# B&R Automation Studio project Cortadora_mappMotion
Automation Studio 4.12.2.93; technology packages: mapp 5.20.0, mappCockpit 5.20.0, mappMotion 5.20.2, mappView 5.20.0

## Configuration AcpTest

CPU 4PPC70.0702-20B, AutomationRuntime B4.91, Build 4.1.2, Safety 0.0, Vc V4.72.9

### Task classes (Cpu.sw)
```
Libraries: NcGlobal, sys_lib, brsystem, runtime
```

### Hardware
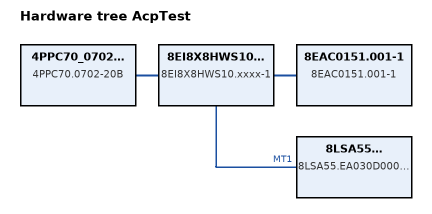
```
4PPC70_0702_20B : 4PPC70.0702-20B v1.5.4.0
  Connector IF2:
    ActivateDevice = 1
  ConfigurationID = Cortadora_mappMotion_AcpTest
  TimerDeviceType = EPLX2X
  TimerDevice = 4PPC70_0702_20B.IF1
  TaskClassIdleTime = 2000
  FileDevice1
  FileDeviceName1 = USER
  FileDevicePath1 = USER_PATH
  KeyMappingFile = VC\4PPC70_0702_20B.dis
8EAC0151.001-1 : 8EAC0151.001-1 v2.2.1.0  [SS -> 8EI8X8HWS10.xxxx-1.SS1]
8EI8X8HWS10.xxxx-1 : 8EI8X8HWS10.xxxx-1 v2.3.1.1  [PLK1 -> 4PPC70_0702_20B.IF1 (NodeNumber=1) [Cable Type=PowerlinkCable, Length=10, Version=1.0.0.3]]
  MotionTP = Acp10Arnc0
  BothEndSwitchesAreNormallyOpen_r1 = on
  QuickStopIsNormallyOpen_r1 = on
8LSA55.EA030D000-1 : 8LSA55.EA030D000-1 v1.0.6.40  [MT -> 8EI8X8HWS10.xxxx-1.MT1]
```

### Acp10cfg.ncc - 4PPC70_0702_20B/Motion/Acp10cfg.ncc
```
NcConfiguration (Version=5.20.1, NcSwId=Acp10)
  ACP10CF1_typ:
    cnt_nettrc_rec_drive = 1500
    bufsize_trace_upload = 1200
    tc_nc_man_task = Cyclic #1
    glob_pv_as_ncobject = Yes
    ncsys_dl_broadcast = Yes
    ncsys_dl_acp_reset = Yes
    safemc_log_err_to_ax = Yes
    network_init:
      ncsw_init_execute = Yes
      automatic_execute = No
      node_nr_warning = Yes
      net_err_before_ncact = Yes
    nettrc:
      enter_parsecrec = Yes
      enter_ncaction = Yes
      save_ring_startidx = Yes
    cam_prof_download:
      cam_dat_dl_parallel = No
      tc_cam_dl_parallel = Task class for NC Manager task
    plk_if[0]:
      if_name = IF1
      tc_CycDat_PLCopen = Task class for NC Manager task
      mc_broadcast_extdat = No
```

### Acp10map.ncm - 4PPC70_0702_20B/Motion/Acp10map.ncm
```
NcMapping (NcSwId=Acp10)
  NcObject gAxis01 (ModuleId=8EI8X8HWS10.xxxx-1, Type=ncAXIS, Channel=1, AcoposSimulation=Off, InitParameter=gAxis01i, AcoposParameter=gAxis01a, Disabled=FALSE, ModuleDisabled=FALSE)
  NcObject 8EI8X8HWS10.xxxx-1_ncV_AXIS1 (ModuleId=8EI8X8HWS10.xxxx-1, Type=ncV_AXIS, Channel=1, Disabled=TRUE, ModuleDisabled=FALSE)
```

## Configuration Config1

CPU 4PPC70.0573-20B, AutomationRuntime B4.91, Build 4.1.2, Safety 0.0, Vc V4.72.6

### Task classes (Cpu.sw)
```
Cyclic#1 (cycle 1600 us, tolerance 0 us):
  MotionCtrl <- MotionCtrl.prg
Cyclic#2 (cycle 11200 us, tolerance 22400 us):
  IMA_Client <- DataHandling.IMA_Client.prg
  VarExchang <- DataHandling.VarExchange.prg
Cyclic#3 (cycle 49600 us, tolerance 49600 us):
  ReadPar <- ReadPar.prg
Cyclic#8 (cycle 9600 us):
  VisuCtrl <- VisuCtrl.prg
DataObjects: DataMap <- DataHandling.DataMap.dob, McAcpSys
NcDataObjects: AcpParTab <- AcpParTab.dob, McDriveLog
VcDataObjects: Visu1 <- Visu.dob
Binaries: vccdt, McAcpSim, vccline, vcfile, arial, vctcal, vccbmp, arsvcreg, vccstr, vcbclass, vccbtn, vcmgr, vcgclass, vcdsint, vcnet, McProfGen, vcchtml, McAcpDrv, vcshared, arflatprv, vccddbox, vcxml, vccnum, vcpdvnc, FWRules, arcoal, vccalarm, vccurl, vcpfar00, vccbar, vcctext, vcpdsw, vcfntttf, vccovl, vccshape, vcalarm, vcpkat, vcctrend, udbdef, vccpopup, vcdsloc, vcrt, TCData, Visu102, Visu101, Visu103, vcpdi815, vcptelo, vcpdihd, vcpk, vcpfppc7, vcpdi855, arconfig, asfw, Cutter, Role, Config_2, ashwd, ExtEncod, iomap, MotionCfg, Config, ashwac, sysconf, User, robot2cm, Visu03, Visu01, Visu02, Visu
Libraries: MpBase, MpAlarmX, astime, runtime, standard, CoTrace, AsZip, FileIO, AsMath, McBase, MpAxis, McPureVAx, McAcpPar, McAcpAx, McAxis, McAxGroup, AsIMA, DataObj, inaclnt, sys_lib, brsystem, asieccon, powerlnk, vcresman, asepl
```

### Hardware
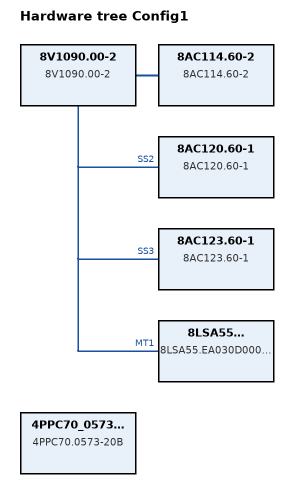
```
4PPC70_0573_20B : 4PPC70.0573-20B v1.5.4.0
  Connector IF1:
    CycleTime = 800
  Connector IF2:
    ActivateDevice = 1
    Mode = Manual
    InternetAddress = 192.168.0.25
    SubnetMask = 255.255.255.0
    Vnc1
    VncVcObjectName1 = Visu1
    VncKeyMappingFile1 = VC\PS2-Keyboard.dis
    ActivateSnmp = 2
  ConfigurationID = Cortadora_mappMotion_Config1
  UserPartitionSize = 0
  RemanentGlobalPvSize = 100
  EnableUsbRemoteInstall = 1
  TimerDeviceType = EPLX2X
  TimerDevice = 4PPC70_0573_20B.IF1
  TaskClassIdleTime = 800
  Cyclic1Duration = 1600
  Cyclic1Tolerance = 0
  Cyclic1Stack = 81920
  Cyclic2Duration = 11200
  Cyclic2Tolerance = 22400
  Cyclic3Duration = 49600
  Cyclic3Tolerance = 49600
  Cyclic8Duration = 9600
  FileDevice1
  FileDeviceName1 = USER
  FileDevicePath1 = USER_PATH
  TimeZone = 45
  ActivateOpcUa = 1
  OpcUaInformationModels_PV_Version = 1
  VcObjectName = Visu1
  KeyMappingFile = VC\4PPC70_0573_20B.dis
8AC114.60-2 : 8AC114.60-2 v1.0.0.8  [SS -> 8V1090.00-2.SS1; PLK1 -> 4PPC70_0573_20B.IF1 (NodeNumber=2) [Cable Type=PowerlinkCable, Length=10, Version=1.0.0.3]]
8AC120.60-1 : 8AC120.60-1 v2.2.0.0  [SS -> 8V1090.00-2.SS2]
  PlugInType = Encoder
  McAcoposTypeID = AcoposPlugInConfig
8AC123.60-1 : 8AC123.60-1 v2.2.0.0  [SS -> 8V1090.00-2.SS3]
  PlugInType = Encoder
  McAcoposTypeID = AcoposPlugInConfig
  LinesPerRevolution = 5000
  IgnoreCheck = 0
8LSA55.EA030D000-1 : 8LSA55.EA030D000-1 v1.0.4.40  [MT -> 8V1090.00-2.MT1]
8V1090.00-2 : 8V1090.00-2 v2.2.0.0
  DriveConfiguration/Module:
    McAcoposTypeID = AcoposConfig
    ActivateACOPOSSimulationOnPLC = 0
  DriveConfiguration/Channel[1]/RealAxis:
    AxisReference = Cutter
    MechanicalElementsIsInvisible = 0
  DriveConfiguration/Channel[1]/RealAxis/MechanicalElements/Gearbox:
    InputIsReadOnly = 0
    Input = 1
    OutputIsReadOnly = 0
    Output = 1
  DriveConfiguration/Channel[1]/RealAxis/MechanicalElements/RotaryToLinearTransformation:
    ReferenceDistanceIsReadOnly = 0
    ReferenceDistance = 1
  DriveConfiguration/Channel[1]/RealAxis/Controller:
    ModeIsReadOnly = 0
    Mode = PositionController
  DriveConfiguration/Channel[1]/RealAxis/Controller/Mode/Position:
    ProportionalGain = 43
    IntegrationTime = 0.0
    PredictionTime = 0.0004
    TotalDelayTime = 0.0004
  DriveConfiguration/Channel[1]/RealAxis/Controller/Mode/Speed:
    ProportionalGainIsReadOnly = 0
    ProportionalGain = 0.4
    IntegrationTimeIsReadOnly = 0
    IntegrationTime = 0.0
    FilterTimeIsReadOnly = 0
    FilterTime = 0.0
  DriveConfiguration/Channel[1]/RealAxis/Controller/Mode/LoopFilters:
    LoopFilterXIsReadOnly = 0
    LoopFilter1 = NotUsed
    LoopFilter2 = NotUsed
    LoopFilter3 = NotUsed
  DriveConfiguration/Channel[1]/RealAxis/Homing:
    ModeIsReadOnly = 0
    Mode = Absolute
  DriveConfiguration/Channel[1]/RealAxis/Homing/Mode:
    Position = -300
  DriveConfiguration/Channel[1]/RealAxis/Homing:
    RestorePositionVariable = 
  DriveConfiguration/Channel[1]/RealAxis/StopReaction:
    QuickstopIsReadOnly = 0
    Quickstop = DecelerationLimit
    DriveErrorIsReadOnly = 0
    DriveError = DecelerationLimit
  DriveConfiguration/Channel[1]/RealAxis/MovementErrorLimits:
    PositionError = 100000000
    VelocityErrorMonitoring = NotUsed
  DriveConfiguration/Channel[1]/RealAxis:
    JerkFilterIsReadOnly = 0
    JerkFilter = NotUsed
  DriveConfiguration/Channel[1]/RealAxis/DigitalInputs/HomingSwitch:
    SourceIsReadOnly = 0
    Source = Force
    Level = High
  DriveConfiguration/Channel[1]/RealAxis/DigitalInputs/PositiveLimitSwitch:
    Source = Force
    Level = High
  DriveConfiguration/Channel[1]/RealAxis/DigitalInputs/NegativeLimitSwitch:
    Source = Force
    Level = High
  DriveConfiguration/Channel[1]/RealAxis/DigitalInputs/Trigger1:
    Source = X1Trigger1
    Level = High
  DriveConfiguration/Channel[1]/RealAxis/DigitalInputs/Trigger2:
    Source = X1Trigger2
    Level = High
  DriveConfiguration/Channel[1]/RealAxis/DigitalInputs/Quickstop:
    Input = NotUsed
  DriveConfiguration/Channel[1]/RealAxis/Simulation:
    SimulationModeOnPLC = SetValueGeneration
    SimulationModeOnACOPOS = NotUsed
  DriveConfiguration/Channel[1]:
    ExternalEncoderAxis = Used
  DriveConfiguration/Channel[1]/ExternalEncoderAxis:
    AxisReference = ExtEncod
  DriveConfiguration/Channel[1]/ExternalEncoderAxis/EncoderLink:
    PositionEncoder = EncoderSS3X11
    PositionFilter = ExtrapolationAndDisturbance
  DriveConfiguration/Channel[1]/ExternalEncoderAxis/EncoderLink/PositionFilter:
    PositionFilterTimeConstant = 0.2
    ExtrapolationTime = 0.1
  DriveConfiguration/Channel[1]/ExternalEncoderAxis:
    MechanicalElementsIsInvisible = 0
  DriveConfiguration/Channel[1]/ExternalEncoderAxis/MechanicalElements/Gearbox:
    InputIsReadOnly = 0
    Input = 1
    OutputIsReadOnly = 0
    Output = 1
  DriveConfiguration/Channel[1]/ExternalEncoderAxis/MechanicalElements/RotaryToLinearTransformation:
    ReferenceDistanceIsReadOnly = 0
    ReferenceDistance = 314.159
  DriveConfiguration/Channel[1]/ExternalEncoderAxis/Homing:
    Mode = Direct
  DriveConfiguration/Channel[1]/ExternalEncoderAxis/Homing/Mode:
    Position = 0.0
    ReferencePulse = NotUsed
  DriveConfiguration/Channel[1]/ExternalEncoderAxis/Homing:
    RestorePositionVariable = 
  DriveConfiguration/Channel[1]/ChannelFeatures:
    FeatureRef[1] = Feature_AcpParTable
```

### Cutter.axis - 4PPC70_0573_20B/mappMotion/Cutter.axis
```
Element Cutter (Type=axis)
  BaseTypeIsReadOnly = 0
  BaseType = RotaryPeriodic
    MeasurementUnitIsReadOnly = 0
    MeasurementUnit = 17476
    MeasurementResolutionIsReadOnly = 0
    MeasurementResolution = 0.01
    CountDirectionIsReadOnly = 0
    CountDirection = Inverse
    PeriodSettings:
      Period = 360.0
  MovementLimitsIsReadOnly = 0
  MovementLimits = Internal
    Position:
      LowerLimitMin = -1.79769313486231E308
      UpperLimitMax = 1.79769313486231E308
      LowerLimit = -1000.0
      UpperLimit = 1000.0
    VelocityIsReadOnly = 0
    Velocity:
      VelocityMax = 3.4E38
      Velocity = 3000000
    AccelerationIsReadOnly = 0
    Acceleration:
      AccelerationMax = 3.4E38
      Acceleration = 5000000000000
    DecelerationIsReadOnly = 0
    Deceleration:
      DecelerationMax = 3.4E38
      Deceleration = 5000000000000
  Alarms = MpAlarmX
```

## Configuration P3wC70

CPU 4PPC70.0702-20B, AutomationRuntime B4.91, Build 4.1.2, Safety 0.0, Vc V4.72.6

### Task classes (Cpu.sw)
```
Cyclic#1 (cycle 1600 us, tolerance 0 us):
  MotionCtrl <- MotionCtrl.prg
  IMA_Client <- DataHandling.IMA_Client.prg
  VarExchang <- DataHandling.VarExchange.prg
Cyclic#3 (cycle 49600 us, tolerance 49600 us):
  ReadPar <- ReadPar.prg
Cyclic#8 (cycle 9600 us):
  VisuCtrl <- VisuCtrl.prg
DataObjects: DataMap <- DataHandling.DataMap.dob, McAcpSys
NcDataObjects: AcpParTab <- AcpParTab.dob, McDriveLog
VcDataObjects: Visu_7 <- Visu_7inch.dob
Binaries: vccdt, vccline, vcfile, vcptelo, vctcal, Visu_702, vccddbox, vccbmp, arsvcreg, vccstr, vcbclass, vccbtn, vcmgr, vcgclass, vcdsint, vcnet, McProfGen, vcchtml, vcpdihd, vcshared, arflatprv, vcxml, vccnum, vcpdvnc, FWRules, vccovl, vcpdi855, arcoal, vccalarm, vccurl, vccbar, vcpfppc7, vcctext, Visu_703, vcpdsw, vcfntttf, McAcpDrv, vccshape, vcalarm, vccpopup, vcpkat, vcctrend, udbdef, vcpdi815, vcdsloc, Visu_701, vcpk, vcrt, TCData, McAcpSim, arial, arconfig, Alarms, asfw, Cutter, Role, ashwd, iomap, MotionCfg, ashwac, sysconf, User, Config_1, ExtEncod, Config_2, Config, robotevi, robot2cm, vcpfar00, Config_4, Virtual
Libraries: MpBase, MpAlarmX, astime, runtime, CoTrace, AsZip, FileIO, asieccon, powerlnk, vcresman, sys_lib, dataobj, asepl, standard, mcbase, mcaxis, mcacpax, mpaxis
```

### Hardware
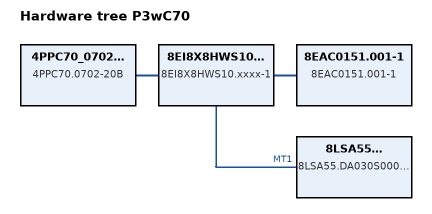
```
4PPC70_0702_20B : 4PPC70.0702-20B v1.5.4.0
  Connector IF1:
    CycleTime = 800
    Mode = CN
    NodeID = 3
    InaNodeNumber = 3
  Connector IF2:
    ActivateDevice = 1
    Mode = Manual
    InternetAddress = 192.168.0.25
    SubnetMask = 255.255.255.0
    Vnc1
    VncVcObjectName1 = Visu_7
    VncKeyMappingFile1 = VC\PS2-Keyboard.dis
    ActivateSnmp = 2
  ConfigurationID = Cortadora_mappMotion_P3
  ConfigVersion = 5.0.0
  UserPartitionSize = 0
  RemanentGlobalPvSize = 1000
  EnableUsbRemoteInstall = 1
  TimerDeviceType = EPLX2X
  TimerDevice = 4PPC70_0702_20B.IF1
  TaskClassIdleTime = 1600
  Cyclic1Duration = 1600
  Cyclic1Tolerance = 0
  Cyclic1Stack = 81920
  Cyclic3Duration = 49600
  Cyclic3Tolerance = 49600
  Cyclic8Duration = 9600
  FileDevice1
  FileDeviceName1 = USER
  FileDevicePath1 = USER_PATH
  VcObjectName = Visu_7
  KeyMappingFile = VC\4PPC70_0702_20B.dis
8EAC0151.001-1 : 8EAC0151.001-1 v2.2.1.0  [SS -> 8EI8X8HWS10.xxxx-1.SS1]
  PlugInType = Encoder
  McAcoposTypeID = AcoposP3PlugInSConfig
  InterfaceType = IncrementalEAC151
  LineResistance = SpecifyValue
  Value = 0.0
  Symmetry = Symmetrical
  LineTermination = 0
  ReferencePulseDetection = 0
  LineCount = 5000
  MaxExpectedOutputFrequency = 200
8EI8X8HWS10.xxxx-1 : 8EI8X8HWS10.xxxx-1 v2.3.1.1  [PLK1 -> 4PPC70_0702_20B.IF1 (NodeNumber=2) [Cable Type=PowerlinkCable, Length=10, Version=1.0.0.3]]
  EnableDNA = on
  DriveConfiguration/Module:
    McAcoposTypeID = AcoposP3DConfig
    ActivateACOPOSSimulationOnPLC = 0
  DriveConfiguration/Encoder/EncoderX41:
    InterfaceType = EnDat
  DriveConfiguration/Channel[1]/RealAxis:
    AxisReference = Cutter
    MechanicalElementsIsInvisible = 0
  DriveConfiguration/Channel[1]/RealAxis/MechanicalElements/Gearbox:
    InputIsReadOnly = 0
    Input = 1
    OutputIsReadOnly = 0
    Output = 1
  DriveConfiguration/Channel[1]/RealAxis/MechanicalElements/RotaryToLinearTransformation:
    ReferenceDistanceIsReadOnly = 0
    ReferenceDistance = 1
  DriveConfiguration/Channel[1]/RealAxis/Controller:
    ModeIsReadOnly = 0
    Mode = PositionControllerWithTorqueFeedForward
  DriveConfiguration/Channel[1]/RealAxis/Controller/Mode/Position:
    ProportionalGainIsReadOnly = 0
    ProportionalGain = 60
    IntegrationTimeIsReadOnly = 0
    IntegrationTime = 0.0
    TotalDelayTime = 0.0004
  DriveConfiguration/Channel[1]/RealAxis/Controller/Mode/Speed:
    ProportionalGainIsReadOnly = 0
    ProportionalGain = 0.9
    IntegrationTimeIsReadOnly = 0
    IntegrationTime = 0.0
    FilterTimeIsReadOnly = 0
    FilterTime = 0.0
  DriveConfiguration/Channel[1]/RealAxis/Controller/Mode:
    FeedForwardIsReadOnly = 0
    FeedForward = Standard
  DriveConfiguration/Channel[1]/RealAxis/Controller/Mode/FeedForward:
    TorqueLoad = 0.0
    TorquePositive = 0.008
    TorqueNegative = 0.00355563
    SpeedTorqueFactor = 0.0109247
    Inertia = 0.00221627
    AccelerationFilterTime = 0.0
  DriveConfiguration/Channel[1]/RealAxis/Controller/Mode/LoopFilters:
    LoopFilterXIsReadOnly = 0
    LoopFilter1 = NotUsed
    LoopFilter2 = NotUsed
    LoopFilter3 = NotUsed
  DriveConfiguration/Channel[1]/RealAxis/Homing:
    ModeIsReadOnly = 0
    Mode = Absolute
  DriveConfiguration/Channel[1]/RealAxis/Homing/Mode:
    Position = -300
  DriveConfiguration/Channel[1]/RealAxis/Homing:
    RestorePositionVariable = 
  DriveConfiguration/Channel[1]/RealAxis/StopReaction:
    QuickstopIsReadOnly = 0
    Quickstop = DecelerationLimit
    DriveErrorIsReadOnly = 0
    DriveError = DecelerationLimit
  DriveConfiguration/Channel[1]/RealAxis/MovementErrorLimits:
    PositionError = 10000
    VelocityErrorMonitoring = NotUsed
  DriveConfiguration/Channel[1]/RealAxis:
    JerkFilterIsReadOnly = 0
    JerkFilter = NotUsed
  DriveConfiguration/Channel[1]/RealAxis/DigitalInputs/HomingSwitch:
    SourceIsReadOnly = 0
    Source = Force
    Level = High
  DriveConfiguration/Channel[1]/RealAxis/DigitalInputs/PositiveLimitSwitch:
    SourceIsReadOnly = 0
    Source = Force
    Level = High
  DriveConfiguration/Channel[1]/RealAxis/DigitalInputs/NegativeLimitSwitch:
    SourceIsReadOnly = 0
    Source = Force
    Level = High
  DriveConfiguration/Channel[1]/RealAxis/DigitalInputs/Trigger1:
    Source = X8Trigger1
    Level = High
  DriveConfiguration/Channel[1]/RealAxis/DigitalInputs/Trigger2:
    Source = X8Trigger2
    Level = High
  DriveConfiguration/Channel[1]/RealAxis/DigitalInputs/Quickstop:
    Input = NotUsed
  DriveConfiguration/Channel[1]/RealAxis/Simulation:
    SimulationModeOnPLC = SetValueGeneration
    SimulationModeOnACOPOS = NotUsed
  DriveConfiguration/Channel[1]:
    ExternalEncoderAxis = Used
  DriveConfiguration/Channel[1]/ExternalEncoderAxis:
    AxisReference = ExtEncod
  DriveConfiguration/Channel[1]/ExternalEncoderAxis/EncoderLink:
    PositionEncoder = EncoderX41x
    PositionFilter = ExtrapolationAndDisturbance
  DriveConfiguration/Channel[1]/ExternalEncoderAxis/EncoderLink/PositionFilter:
    PositionFilterTimeConstant = 0.0
    ExtrapolationTime = 0.1
  DriveConfiguration/Channel[1]/ExternalEncoderAxis:
    MechanicalElementsIsInvisible = 0
  DriveConfiguration/Channel[1]/ExternalEncoderAxis/MechanicalElements/Gearbox:
    InputIsReadOnly = 0
    Input = 1
    OutputIsReadOnly = 0
    Output = 1
  DriveConfiguration/Channel[1]/ExternalEncoderAxis/MechanicalElements/RotaryToLinearTransformation:
    ReferenceDistanceIsReadOnly = 0
    ReferenceDistance = 31.4159
  DriveConfiguration/Channel[1]/ExternalEncoderAxis/Homing:
    Mode = Direct
  DriveConfiguration/Channel[1]/ExternalEncoderAxis/Homing/Mode:
    Position = 0.0
    ReferencePulse = NotUsed
  DriveConfiguration/Channel[1]/ExternalEncoderAxis/Homing:
    RestorePositionVariable = 
8LSA55.DA030S000-3 : 8LSA55.DA030S000-3 v2.2.0.1  [MT -> 8EI8X8HWS10.xxxx-1.MT1]
  M1/MotorParameters:
    MOTOR_AMB_TEMP_RATED = 40
```

### ExtEncod.axis - 4PPC70_0702_20B/mappMotion/ExtEncod.axis
```
Element ExtEncod (Type=axis)
  BaseTypeIsReadOnly = 0
  BaseType = Linear
    MeasurementUnit = 5066068
    MeasurementResolutionIsReadOnly = 0
    MeasurementResolution = 0.01
    CountDirectionIsReadOnly = 0
    CountDirection = Inverse
  MovementLimitsIsReadOnly = 0
  MovementLimits = Internal
    Position:
      LowerLimitMin = -1.79769313486231E308
      UpperLimitMax = 1.79769313486231E308
      LowerLimit = -1000.0
      UpperLimit = 1000.0
    VelocityIsReadOnly = 0
    Velocity:
      VelocityMax = 3.4E38
      Velocity = 1000
    AccelerationIsReadOnly = 0
    Acceleration:
      AccelerationMax = 3.4E38
      Acceleration = 10000
    DecelerationIsReadOnly = 0
    Deceleration:
      DecelerationMax = 3.4E38
      Deceleration = 10000
  Alarms = MpAlarmX
```

### MotionCfg.mappmotioncfg - 4PPC70_0702_20B/mappMotion/MotionCfg.mappmotioncfg
```
Element MappMotionConfiguration (Type=mappmotioncfg)
  Processing:
    ProcessingTaskClass = 1
  SharedAlarms:
    Axis = MpAlarmX
```

## Logical view

Binary libraries used (declarations not repeated): operator, runtime, astime, AsIecCon, standard, AsZip, FileIO, AsMath, NcGlobal 5.20.1, sys_lib, brsystem, MpBase, MpAlarmX 5.20.0, CoTrace, McBase, MpAxis, McPureVAx 5.20.2, McAcpPar 5.20.2, McAcpAx, McAxis, McAxGroup 5.20.2, AsIMA, DataObj, inaclnt

### Global.typ - Global data types
```iecst
TYPE
	gCutter_enum :
		(
		Default,
		Encoder,
		Time,
		Sensor,
		Speed,
		EncoderDieCutter,
		SensorDieCutter
		);
	DataCollector_state_enum :
		(
		ST_IDLE,
		ST_CONNECTING,
		ST_CONNECTED,
		ST_CLOSE_CONNECTION,
		ST_ERROR_ACTIVE,
		ST_RESET_ERROR
		);
END_TYPE
```

### Global.var - Global variables
```iecst
VAR
	MODE_SELECTED : gCutter_enum;
	posTroqueladora : LREAL;
	SensorSignal : BOOL;
	MachineStateIndex : UINT := 0;
	MachineInOperation : BOOL;
	MachineInitializing : BOOL;
	MachineAutotuning : BOOL;
	MachineHoming : BOOL;
	MachineReady : BOOL;
	CurrentPage : INT;
END_VAR
VAR RETAIN
	HMI_MODE_SELECTED : gCutter_enum;
END_VAR
VAR
	TotalCutsPerMode : LREAL;
	BoxIsOpen : BOOL;
	CycleTime : REAL := 1.6;
	MinuteInMiliseconds : DINT := 60000;
	CycleTimeSum : REAL;
	CutsPerMinute_Distance : REAL;
	CutsPerMinute_Time : REAL;
	CutsPerMinute_Sensor : REAL;
	cutEnabled : BOOL; (*Info proveniente de la troqueladora*)
	auxToCut : BOOL;
	encActPosPerRev : DINT;
	actPosExtEncoder : LREAL; (*Info proveniente de la troqueladora*)
	oneCutEncoderCutterDieCmd : BOOL;
END_VAR
```


### Program Logical/MotionCtrl (IEC)

#### Main.st - Init, cyclic, exit code
```iecst
PROGRAM _INIT
	(* Insert code here *)
	MpAxisBasic_Cutter.MpLink := ADR(Cutter);
	MpAxisBasic_Cutter.Parameters := ADR(MpAxisBasicPar_Cutter);

	MpAxisBasicPar_Cutter.Velocity := DefaultVelocity;
	MpAxisBasicPar_Cutter.Acceleration := DefaultAcceleration;
	MpAxisBasicPar_Cutter.Deceleration := DefaultDeceleration;
	MpAxisBasicPar_Cutter.Distance := DefaultDistance;
	MpAxisBasicPar_Cutter.Position := DefaultPosition;

	MC_BR_InitHome_AcpAx_0.Axis := ADR(Cutter);
	MC_BR_InitHome_AcpAx_0.HomingParameters := McAcpAxHomingPar_0;
	McAcpAxHomingPar_0.HomingMode := InitHomingMode;

	MC_BR_InitHome_AcpAx_0.Axis := ADR(Cutter);
	MC_BR_InitHome_AcpAx_0.HomingParameters.HomingMode := InitHomingMode;
	MC_BR_InitHome_AcpAx_0.HomingParameters.Position := DefaultPosition;
	MC_BR_InitHome_AcpAx_0.HomingParameters.StartVelocity := 50;
	MC_BR_InitHome_AcpAx_0.HomingParameters.HomingVelocity := 50;
	MC_BR_InitHome_AcpAx_0.HomingParameters.Acceleration := 500;
	MC_BR_InitHome_AcpAx_0.HomingParameters.SwitchEdge := 0;
	MC_BR_InitHome_AcpAx_0.HomingParameters.StartDirection := 1;
	MC_BR_InitHome_AcpAx_0.HomingParameters.HomingDirection := 0;

	MpAxisBasicPar_Cutter.Homing.Mode := HomingMode;
	MpAxisBasicPar_Cutter.Homing.Position := DefaultPosition;

	//Autotune settings
	MpAxisBasicPar_Cutter.AutoTune.MaxCurrentPercent := 75;
	MpAxisBasicPar_Cutter.AutoTune.MaxDistance := 5;
	MpAxisBasicPar_Cutter.AutoTune.MaxPositionError := 2000;

	(*//Reading external encoder
	MC_BR_CyclicProcessParID_AcpAx_0.Axis := ADR(ExtEncod);
	MC_BR_CyclicProcessParID_AcpAx_0.DataAddress := ADR(McAcpAxCycParID_0);
	MC_BR_CyclicProcessParID_AcpAx_0.Mode := mcACPAX_CYCLIC_PARID_READ;
	MC_BR_CyclicProcessParID_AcpAx_0.NumberOfParIDs := 1;

	McAcpAxCycParID_0.DataType:= mcACPAX_PARTYPE_DINT;
	McAcpAxCycParID_0.ParID := 246;//423 Actual Position, 246 Actual Position per Revolution
	McAcpAxCycParID_0.RefreshMode := mcACPAX_CYCLIC_EVERY_RECORD;
	McAcpAxCycParID_0.VariableAddress := ADR(EncoderActPos);*)

	MpAxisBasic_Cutter.Enable := TRUE;

END_PROGRAM

PROGRAM _CYCLIC

	Pulses := REAL_TO_UINT(HMIPulses * 4);

	vAxisEncoderActPos;
	//Basic calculation of encoder perimeter adjusted via HMI
	EncoderPerimeter := (amPI * EncoderDiameter);

	//Cutting Offset - Not used
	DelayTimer_0.PT := UDINT_TO_TIME(SensorCutDelay);

	//mapping for visu
	BoxIsOpen := NOT MpAxisBasic_Cutter.Info.DigitalInputsStatus.DriveEnable;

	CASE MODE_SELECTED OF

		Default:

			InitAxis;

			CutterTimer.IN := FALSE;
			CutterTimer.PT := DINT_TO_TIME(0);

		Encoder:

			MpAxisBasicPar_Cutter.Velocity := DefaultVelocity;
			MpAxisBasicPar_Cutter.Acceleration := DefaultAcceleration;
			MpAxisBasicPar_Cutter.Deceleration := DefaultDeceleration;

			//Start Encoder Position Reading
			//MC_BR_CyclicProcessParID_AcpAx_0.Enable := TRUE;
			//EncoderActPos := encActPosPerRev;
			encActPosPerRev;

			IF CorrectDistance THEN
				ActualProductLength := HMICuttingLength + (CuttingOffset *-1);
				CorrectionFactor := (HMICuttingLength/ActualProductLength);
				HMICorrectionFactorPercentage := (CorrectionFactor *100) - 100;
				CuttingOffset := 0;
				CorrectDistance := FALSE;
			END_IF;

			HMICorrectionFactorMilimeters :=((HMICorrectionFactorPercentage/100) * HMICuttingLength);

			IF ClockwiseCount THEN

				IF EDGEPOS(EncoderActPosOld > EncoderActPos) AND ((EncoderActPosOld - EncoderActPos) > (Pulses*0.995)) THEN
					FullTurnCount := FullTurnCount + 1;
				END_IF;

				PartOfTurn := (DINT_TO_REAL(EncoderActPos)/Pulses);

			ELSE

				IF EDGEPOS(EncoderActPos > EncoderActPosOld) AND ((EncoderActPos - EncoderActPosOld) > (Pulses*0.995)) THEN
					FullTurnCount := FullTurnCount + 1;
				END_IF;

				PartOfTurn := 1 - (DINT_TO_REAL(EncoderActPos)/Pulses);

			END_IF;

			IF PartOfTurn >= (0.99) OR PartOfTurn < 0 THEN
				PartOfTurn := 0;
			END_IF;

			RealTurns := FullTurnCount + PartOfTurn;

			IF Empezar AND cutEnabled THEN

				MachineInOperation := TRUE;

				CycleTimeSum := CycleTimeSum + CycleTime;

				CountTurns;

				IF MpAxisBasic_Cutter.MoveDone THEN
					MpAxisBasic_Cutter.MoveAdditive := FALSE;
				END_IF;

				IF EDGEPOS(MpAxisBasic_Cutter.MoveDone) THEN
					NumberOfCuts_Distance := NumberOfCuts_Distance + 1;
				END_IF;

				RemainingDistance := ((NeededTurns - RealTurns) * EncoderPerimeter);
				TraveledDistance := HMICuttingLength - RemainingDistance;

				HMITraveledDistance := TraveledDistance ;
				HMIRemainingDistance := RemainingDistance;

				MC_BR_CyclicProcessParID_AcpAx_0();

				IF MpAxisBasic_Cutter.Error THEN
					MpAxisBasic_Cutter.MoveAdditive := FALSE;
					MpAxisBasic_Cutter.ErrorReset := TRUE;
				ELSE
					MpAxisBasic_Cutter.ErrorReset := FALSE;
				END_IF;

			END_IF;

			IF NOT Empezar THEN

				HMITraveledDistance := 0 ;
				HMIRemainingDistance := 0;
				CurrentProductTurns := 0;
				NeededTurns := 0;

				MC_BR_CyclicProcessParID_AcpAx_0.Enable := FALSE;

			END_IF;

			TotalCutsPerMode := NumberOfCuts_Distance;

		Time:

			MpAxisBasicPar_Cutter.Velocity := DefaultVelocity;
			MpAxisBasicPar_Cutter.Acceleration := DefaultAcceleration;
			MpAxisBasicPar_Cutter.Deceleration := DefaultDeceleration;

			CycleTimeSum := CycleTimeSum + CycleTime;

			IF Empezar THEN

				MachineInOperation := TRUE;
				CycleTimeSum := CycleTimeSum + CycleTime;
				UserTime := REAL_TO_DINT(HMITime*1000);
				TimeIsOver := CutterTimer.Q;
				CutterTimer.PT := DINT_TO_TIME(UserTime);
				ElapsedTime := (TIME_TO_REAL(CutterTimer.ET)/1000);
				RemainingTime := (REAL_TO_DINT(HMITime) - ElapsedTime);

				IF TimeIsOver THEN
					DelayTimer_0.IN := TRUE;
					CutterTimer.IN := FALSE;
				ELSE
					CutterTimer.IN := TRUE;
				END_IF;

				IF MpAxisBasic_Cutter.MoveDone THEN
					MpAxisBasic_Cutter.MoveAdditive := FALSE;
				END_IF;

				IF EDGEPOS(MpAxisBasic_Cutter.MoveDone) THEN
					NumberOfCuts_Time := NumberOfCuts_Time + 1;
				END_IF;

			ELSE

				ElapsedTime := 0;
				RemainingTime := 0;

			END_IF;

			TotalCutsPerMode := NumberOfCuts_Time;
			CutsPerMinute_Time := (60/HMITime);

			CutterTimer();

		Sensor:

			MpAxisBasicPar_Cutter.Velocity := DefaultVelocity;
			MpAxisBasicPar_Cutter.Acceleration := DefaultAcceleration;
			MpAxisBasicPar_Cutter.Deceleration := DefaultDeceleration;

			CycleTimeSum := CycleTimeSum + CycleTime;

			IF Empezar AND cutEnabled THEN

				MachineInOperation := TRUE;
				SensorSignal := MpAxisBasic_Cutter.Info.DigitalInputsStatus.Trigger1;
				FilterTimer_0.PT := UINT_TO_TIME(FilterTime);

				IF NOT FilterActive THEN

					IF EDGEPOS(MpAxisBasic_Cutter.Info.DigitalInputsStatus.Trigger1 OR inputTest) OR auxToCut THEN
						auxToCut := FALSE;
						FilterTimer_0.IN := TRUE;
						DelayTimer_0.IN := TRUE;
						FilterActive := TRUE;
					END_IF;

				END_IF;

				IF FilterTimer_0.Q THEN
					FilterActive := FALSE;
					FilterTimer_0.IN := FALSE;
				END_IF;

				FilterActive := FilterTimer_0.IN;

				FilterTimer_0();

				IF MpAxisBasic_Cutter.MoveDone THEN
					MpAxisBasic_Cutter.MoveAdditive := FALSE;
					SensorSignal := FALSE;
				END_IF;

				IF EDGEPOS(MpAxisBasic_Cutter.MoveDone) THEN
					NumberOfCuts_Sensor := NumberOfCuts_Sensor + 1;
				END_IF;

			END_IF;

			TotalCutsPerMode := NumberOfCuts_Sensor;
			CutsPerMinute_Sensor := NumberOfCuts_Sensor/CycleTimeSum;
		Speed:

			MachineInOperation := TRUE;

			CycleTimeSum := CycleTimeSum + CycleTime;

			IF Empezar THEN

				MpAxisBasicPar_Cutter.Velocity := HMIRevolutionsPerSecond * UnitsPerRevolution;
				MpAxisBasicPar_Cutter.Acceleration := MpAxisBasicPar_Cutter.Velocity * 10;
				MpAxisBasicPar_Cutter.Deceleration := MpAxisBasicPar_Cutter.Velocity * 10;
				MpAxisBasic_Cutter.MoveVelocity := TRUE;

			ELSE

				IF NOT MpAxisBasic_Cutter.IsHomed THEN
					ManualMoveAbsolute := TRUE;
				END_IF;

				MpAxisBasic_Cutter.MoveVelocity := FALSE;

			END_IF;

			IF (MpAxisBasic_Cutter.Velocity <> MpAxisBasicPar_Cutter.Velocity) AND Empezar THEN
				MpAxisBasic_Cutter.Update := TRUE;
			END_IF;

			IF MpAxisBasic_Cutter.UpdateDone THEN
				MpAxisBasic_Cutter.Update := FALSE;
			END_IF;

	END_CASE;

	//Whenever the operator presses Manual Cut the motor should do a full turn unless there is an active movement
	IF ManualCut AND (MpAxisBasic_Cutter.Info.PLCopenState = AxisStandstill) THEN

		MpAxisBasic_Cutter.MoveAdditive := TRUE;

		IF MpAxisBasic_Cutter.MoveDone THEN
			MpAxisBasic_Cutter.MoveAdditive := FALSE;
			ManualCut := FALSE;
		END_IF;

	END_IF;

	//For Visu
	IF Empezar THEN

		Count := Count + 0.0016;
		IF CountOld > Count THEN
			MaxCount := CountOld;
		END_IF;

		CountOld := Count;

	ELSE

		MachineInOperation := FALSE;
		MpAxisBasic_Cutter.MoveVelocity := FALSE;
		MpAxisBasic_Cutter.MoveAdditive := FALSE;
		CycleTimeSum := 0;
		MaxCount := 0;
		Count := 0;

	END_IF;

	//Sum of total cuts
	IF EDGEPOS(MpAxisBasic_Cutter.MoveDone) THEN

		Count := 0;
		TotalCuts := TotalCuts + 1;

	END_IF;

	IF MaxCount = 0 THEN
		ProductionSpeed := 0;
	ELSE
		ProductionSpeed := 60/MaxCount;
	END_IF;

	TotalCurrentCuts := NumberOfCuts_Time + NumberOfCuts_Sensor + NumberOfCuts_Distance;

	IF ResetCutsPerMode THEN
		NumberOfCuts_Time := 0;
		NumberOfCuts_Sensor := 0;
		NumberOfCuts_Distance := 0;
		ResetCutsPerMode := FALSE;
	END_IF;

	IF ResetTotalCuts THEN

		TotalCuts := 0;
		ResetTotalCuts := FALSE;

	END_IF;

	//Manual Controls
	IF NOT Empezar AND NOT MpAxisBasic_Cutter.MoveActive AND (CurrentPage = 1) THEN

		IF ManualMoveAdditivePos THEN
			ManualMoveAdditivePos := FALSE;
			MpAxisBasic_Cutter.MoveAdditive := TRUE;
			MpAxisBasicPar_Cutter.Distance := HMIDistance;
		END_IF;

		IF ManualMoveAdditiveNeg THEN
			ManualMoveAdditiveNeg := FALSE;
			MpAxisBasic_Cutter.MoveAdditive := TRUE;
			MpAxisBasicPar_Cutter.Distance := HMIDistance * -1;
		END_IF;

		IF ManualMoveAbsolute THEN
			MpAxisBasic_Cutter.MoveAbsolute := TRUE;
			MpAxisBasicPar_Cutter.Position := HomePosition;
			MpAxisBasicPar_Cutter.Direction := 0;
		END_IF;

	END_IF;

	IF MpAxisBasic_Cutter.MoveDone THEN

		ManualMoveAdditivePos := FALSE;
		ManualMoveAdditiveNeg := FALSE;
		ManualMoveAbsolute := FALSE;
		MpAxisBasic_Cutter.MoveAdditive := FALSE;
		MpAxisBasic_Cutter.MoveAbsolute := FALSE;

	END_IF;

	IF DelayTimer_0.Q THEN

		DelayTimer_0.IN := FALSE;
		//MpAxisBasic_Cutter.MoveAdditive := TRUE;

	END_IF;

	IF (CurrentPage = 0) THEN

		MpAxisBasicPar_Cutter.Distance := DefaultDistance;
		MpAxisBasicPar_Cutter.Position := DefaultPosition;

	END_IF;

	IF NOT MpAxisBasic_Cutter.Info.DigitalInputsStatus.DriveEnable THEN

		Empezar := FALSE;
		MpAxisBasic_Cutter.Power := FALSE;
		MpAxisBasic_Cutter.Home := FALSE;
		MpAxisBasic_Cutter.MoveAdditive := FALSE;
		MpAxisBasic_Cutter.MoveAbsolute := FALSE;
		MpAxisBasic_Cutter.MoveVelocity := FALSE;
		ManualMoveAdditivePos := FALSE;
		ManualMoveAdditiveNeg := FALSE;
		ManualMoveAbsolute := FALSE;
		MODE_SELECTED := Default;

	ELSE

		MpAxisBasic_Cutter.Stop := FALSE;

	END_IF;

	IF MpAxisBasic_Cutter.Error THEN
		MpAxisBasic_Cutter.ErrorReset := TRUE;
	ELSE
		MpAxisBasic_Cutter.ErrorReset := FALSE;
	END_IF;

	IF Empezar THEN
		OperationSignal := OperationSignal + CycleTime;
		IF (OperationSignal >= (CycleTime * 625)) THEN
			IF OperationSignalOut = 1 THEN
				OperationSignalOut := 0;
			ELSE
				OperationSignalOut := 1;
			END_IF;
			OperationSignal := 0;
		END_IF;
	ELSE
		OperationSignalOut := 1;
	END_IF;

	IF CycleTimeSum >= MinuteInMiliseconds THEN
		CycleTimeSum := 0;
	END_IF;

	//Auxiliar para hacer un primer corte cuando se habilite desde la troqueladora
	IF NOT(cutEnabled) THEN
		auxToCut := TRUE;
	END_IF;

	DelayTimer_0();
	MpAxisBasic_Cutter();

END_PROGRAM

PROGRAM _EXIT

	MpAxisBasic_Cutter.Enable := FALSE;
	MpAxisBasic_Cutter();

END_PROGRAM
```

#### Variables.var - Local variables
```iecst
(*Time Mode*)
VAR
	TimeIsOver : BOOL;
	CutterTimer : TON;
	UserTime : DINT;
END_VAR
VAR RETAIN
	HMITime : REAL := 1;
END_VAR
VAR
	NumberOfCuts_Time : LREAL;
	ElapsedTime : REAL;
	RemainingTime : REAL;
END_VAR
(*Cutter*)
VAR
	MpAxisBasic_Cutter : MpAxisBasic;
	MpAxisBasicPar_Cutter : MpAxisBasicParType;
	MC_BR_ProcessParID_AcpAx_0 : MC_BR_ProcessParID_AcpAx;
	ParID_FB_Mode : McAcpAxProcessParIDModeEnum;
	InitHomingMode : McHomingModeEnum := mcHOMING_ABSOLUTE;
	HomingMode : McHomingModeEnum := mcHOMING_ABSOLUTE;
	McAcpAxProcessParIDType_0 : McAcpAxProcessParIDType;
END_VAR
VAR CONSTANT
	DefaultPosition : LREAL := 0.00;
	DefaultVelocity : REAL := 65000;
	DefaultDistance : LREAL := 360;
	DefaultAcceleration : REAL := DefaultVelocity * 10;
	DefaultDeceleration : REAL := DefaultVelocity * 10;
END_VAR
VAR
	NoHome : BOOL;
	ReadyToHome : BOOL;
	ReadyToInitHome : BOOL;
	ReadyToPower : BOOL;
	MC_BR_InitHome_AcpAx_0 : MC_BR_InitHome_AcpAx;
	McAcpAxHomingPar_0 : McAcpAxHomingParType;
END_VAR
(*Set Voltage*)
VAR
	BusVoltage : REAL := 325;
	SetVoltage : BOOL;
END_VAR
(*Read Encoder 2 Actual Position*)
VAR
	MC_BR_CyclicProcessParID_AcpAx_0 : MC_BR_CyclicProcessParID_AcpAx;
	McAcpAxCycParID_0 : McAcpAxCycParIDType;
	MaxThreshold : UINT := 18000;
	MinThreshold : UINT := 2000;
	StartCount : BOOL;
	MaxCount : REAL;
	CountOld : REAL;
	Count : REAL;
	RealTurns : REAL;
	CurrentProductTurns : REAL;
	NeededTurnsOld : REAL;
	NeededTurns : REAL;
	ExceededPart : DINT;
	PartOfTurn : REAL;
	FullTurnIncrements : UINT := 20000;
	FullTurnCount : REAL;
	EncoderActPosOld : DINT;
	EncoderActPos : DINT;
	ReadEncoder : BOOL;
	Empezar : BOOL; (*AutoStart*)
	vAxisEncoderActPos : DINT;
END_VAR
(*Distance Mode (Encoder 2)*)
VAR RETAIN
	HMICuttingLength : REAL := 314.159; (*in mm*)
END_VAR
VAR
	ActualProductLength : REAL;
	EncoderPerimeter : REAL := 314.159265; (*in mm*)
END_VAR
VAR RETAIN
	EncoderDiameter : REAL := 100; (*in mm*)
END_VAR
VAR
	CorrectDistance : BOOL;
END_VAR
VAR RETAIN
	HMICorrectionFactorMilimeters : REAL;
	HMICorrectionFactorPercentage : REAL;
	CorrectionFactor : REAL := 1; (*Value to counter phsysical deviations between machines. Adjust as necessary. Value used in Acopos 1090 0.9957 *)
END_VAR
VAR
	NumberOfCuts_Distance : LREAL;
	HMIRelativeDistanceOld : REAL;
	RelativeDistanceOld : REAL;
	HMIRelativeDistance : REAL;
	RelativeDistance : REAL;
	HMITraveledDistance : REAL;
	TraveledDistance : REAL;
	HMIRemainingDistance : REAL;
	RemainingDistance : REAL;
END_VAR
VAR RETAIN
	CuttingOffset : REAL;
END_VAR
VAR
	CalculatedProductSpeed : REAL;
END_VAR
VAR RETAIN
	ClockwiseCount : BOOL := TRUE;
END_VAR
(*Write encoder 2 values*)
VAR
	MC_BR_ProcessParID_AcpAx_1 : MC_BR_ProcessParID_AcpAx;
	McAcpAxProcessParIDType_1 : McAcpAxProcessParIDType;
	LoadUnits : UDINT := 5000;
	MC_BR_ProcessParID_AcpAx_2 : MC_BR_ProcessParID_AcpAx;
	McAcpAxProcessParIDType_2 : McAcpAxProcessParIDType;
	Proportion : REAL := 0.6;
END_VAR
VAR RETAIN
	HMIPulses : REAL := 5000;
END_VAR
VAR
	Pulses : UINT := 20000;
	AxisDisabled : McAxisPLCopenStateEnum := mcAXIS_DISABLED;
	AxisStandstill : McAxisPLCopenStateEnum := mcAXIS_STANDSTILL;
END_VAR
(*Manual Controls*)
VAR
	ManualCut : BOOL;
	ManualMoveAdditiveNeg : BOOL;
	ManualMoveAdditivePos : BOOL;
	ManualMoveAbsolute : BOOL;
	ManualMoveVelocity : BOOL;
END_VAR
VAR RETAIN
	HomePosition : LREAL := 60;
END_VAR
VAR
	HMIVelocity : REAL := 65000;
	HMIDistance : LREAL := 10;
END_VAR
(* Sensor Mode*)
VAR
	RPM : DINT;
	Torque : REAL;
	ProductionSpeed : REAL;
	MC_BR_CyclicProcessParID_AcpAx_1 : MC_BR_CyclicProcessParID_AcpAx;
	McAcpAxCycParID_1 : McAcpAxCycParIDType;
	MC_BR_CyclicProcessParID_AcpAx_2 : MC_BR_CyclicProcessParID_AcpAx;
	McAcpAxCycParID_2 : McAcpAxCycParIDType;
	MC_BR_CyclicProcessParID_AcpAx_3 : MC_BR_CyclicProcessParID_AcpAx;
	McAcpAxCycParID_3 : McAcpAxCycParIDType;
	NumberOfCuts_Sensor : REAL;
	SensorCutDelay : UDINT := 0;
	DelayTimer_0 : TON;
	FilterTimer_0 : TON;
	FilterActivated : BOOL;
	TimerStopped : TIME;
END_VAR
VAR RETAIN
	FilterTime : UINT;
END_VAR
VAR
	FilteredCut : BOOL;
	inputTest : BOOL;
	FilterActive : BOOL;
END_VAR
(*Misc*)
VAR
	TotalCurrentCuts : LREAL;
END_VAR
VAR RETAIN
	TotalCuts : REAL;
END_VAR
VAR
	ResetCutsPerMode : BOOL;
	ResetTotalCuts : BOOL;
	ParameterReading : ParameterReading_enum;
	ParCount : USINT;
	OperationSignal : REAL;
	OperationSignalOut : USINT;
	ReadParID : BOOL;
	MotorTorque : UINT := 277;
END_VAR
(*Speed Mode*)
VAR RETAIN
	HMIRevolutionsPerSecond : REAL := 1;
END_VAR
VAR
	UnitsPerRevolution : REAL := 360;
END_VAR
```

#### Types.typ - Local data types
```iecst
TYPE
	ParameterReading_enum :
		(
		RESET,
		TORQUE,
		REVS_PER_MINUTE,
		PRODUCTION_SPEED
		);
END_TYPE
```

#### SetParIDs.st
```iecst
ACTION InitParIDWrite:

	MpAxisBasic_Cutter.Enable := FALSE;
	//Write encoder values

	//Bus voltage
	MC_BR_ProcessParID_AcpAx_0.Axis := ADR(Cutter);
	MC_BR_ProcessParID_AcpAx_0.Execute := TRUE;
	MC_BR_ProcessParID_AcpAx_0.DataAddress := ADR(McAcpAxProcessParIDType_0);
	MC_BR_ProcessParID_AcpAx_0.NumberOfParIDs := 1;
	MC_BR_ProcessParID_AcpAx_0.Mode := mcACPAX_PARID_SET;

	McAcpAxProcessParIDType_0.DataType := mcACPAX_PARTYPE_REAL;
	McAcpAxProcessParIDType_0.ParID := 390;
	McAcpAxProcessParIDType_0.VariableAddress := ADR(BusVoltage);

	//Scale Units
	MC_BR_ProcessParID_AcpAx_1.Axis := ADR(extEncod);
	MC_BR_ProcessParID_AcpAx_1.Execute := TRUE;
	MC_BR_ProcessParID_AcpAx_1.DataAddress := ADR(McAcpAxProcessParIDType_0);
	MC_BR_ProcessParID_AcpAx_1.NumberOfParIDs := 1;
	MC_BR_ProcessParID_AcpAx_1.Mode := mcACPAX_PARID_SET;

	McAcpAxProcessParIDType_1.DataType := mcACPAX_PARTYPE_UDINT;
	McAcpAxProcessParIDType_1.ParID := 420;
	McAcpAxProcessParIDType_1.VariableAddress := ADR(LoadUnits);

	//Pulses
	MC_BR_ProcessParID_AcpAx_2.Axis := ADR(extEncod);
	MC_BR_ProcessParID_AcpAx_2.Execute := TRUE;
	MC_BR_ProcessParID_AcpAx_2.DataAddress := ADR(McAcpAxProcessParIDType_0);
	MC_BR_ProcessParID_AcpAx_2.NumberOfParIDs := 1;
	MC_BR_ProcessParID_AcpAx_2.Mode := mcACPAX_PARID_SET;

	McAcpAxProcessParIDType_2.DataType := mcACPAX_PARTYPE_UDINT;
	McAcpAxProcessParIDType_2.ParID := 289;
	McAcpAxProcessParIDType_2.VariableAddress := ADR(Pulses);

	IF MC_BR_ProcessParID_AcpAx_0.Done AND MC_BR_ProcessParID_AcpAx_1.Done AND MC_BR_ProcessParID_AcpAx_2.Done THEN

		MC_BR_ProcessParID_AcpAx_0.Execute := FALSE;
		MC_BR_ProcessParID_AcpAx_1.Execute := FALSE;
		MC_BR_ProcessParID_AcpAx_2.Execute := FALSE;
		InitWrite := FALSE;

	END_IF;

	MC_BR_ProcessParID_AcpAx_0();
	MC_BR_ProcessParID_AcpAx_1();
	MC_BR_ProcessParID_AcpAx_2();

END_ACTION
```

#### GetParIDs.st
```iecst
ACTION ReadParIDs:

	CASE ParameterReading OF
		RESET:
			MC_BR_CyclicProcessParID_AcpAx_1.Enable := FALSE;
			MC_BR_CyclicProcessParID_AcpAx_1();
			IF ParCount = 0 THEN
				ParameterReading := TORQUE;
				ParCount := ParCount + 1;
			ELSIF ParCount = 1 THEN
				ParameterReading := REVS_PER_MINUTE;
				ParCount := ParCount + 1;
			ELSIF ParCount = 2 THEN
				(*ParameterReading := PRODUCTION_SPEED;*)
				ParCount := 0(*ParCount + 1*);
			ELSIF ParCount = 3 THEN
				ParCount :=0;
			END_IF;

		TORQUE:
			McAcpAxCycParID_1.ParID := MotorTorque;
			McAcpAxCycParID_1.VariableAddress := ADR(Torque);
			McAcpAxCycParID_1.DataType:= mcACPAX_PARTYPE_DINT;
			ParCount:= 1;
			ParameterReading := RESET;
		REVS_PER_MINUTE:
			McAcpAxCycParID_1.ParID := 298(*331*);
			McAcpAxCycParID_1.VariableAddress := ADR(RPM);
			McAcpAxCycParID_1.DataType:= mcACPAX_PARTYPE_DINT;
			ParCount:= 2;
			ParameterReading := RESET;
		PRODUCTION_SPEED:
			McAcpAxCycParID_1.ParID := 7760;
			McAcpAxCycParID_1.VariableAddress := ADR(ProductionSpeed);
			McAcpAxCycParID_1.DataType:= mcACPAX_PARTYPE_REAL;
			ParCount:= 3;
			ParameterReading := RESET;
	END_CASE;

	MC_BR_CyclicProcessParID_AcpAx_1.Enable := TRUE;
	MC_BR_CyclicProcessParID_AcpAx_1.Axis := ADR(Cutter);
	MC_BR_CyclicProcessParID_AcpAx_1.DataAddress := ADR(McAcpAxCycParID_1);
	MC_BR_CyclicProcessParID_AcpAx_1.Mode := mcACPAX_CYCLIC_PARID_READ;
	MC_BR_CyclicProcessParID_AcpAx_1.NumberOfParIDs := 1;

	McAcpAxCycParID_1.DataType:= mcACPAX_PARTYPE_DINT;
	McAcpAxCycParID_1.RefreshMode := mcACPAX_CYCLIC_EVERY_RECORD;

	MC_BR_CyclicProcessParID_AcpAx_1();

//	McAcpAxCycParID_1.ParID := MotorTorque;//423 Actual Position, 246 Actual Position per Revolution
//	McAcpAxCycParID_1.VariableAddress := ADR(Torque);
//	MC_BR_CyclicProcessParID_AcpAx_2.Enable := TRUE;
//	MC_BR_CyclicProcessParID_AcpAx_2.Axis := ADR(Cutter);
//	MC_BR_CyclicProcessParID_AcpAx_2.DataAddress := ADR(McAcpAxCycParID_2);
//	MC_BR_CyclicProcessParID_AcpAx_2.Mode := mcACPAX_CYCLIC_PARID_READ;
//	MC_BR_CyclicProcessParID_AcpAx_2.NumberOfParIDs := 1;
//
//	McAcpAxCycParID_2.DataType:= mcACPAX_PARTYPE_DINT;
//	McAcpAxCycParID_2.ParID := 331;//423 Actual Position, 246 Actual Position per Revolution
//	McAcpAxCycParID_2.RefreshMode := mcACPAX_CYCLIC_EVERY_RECORD;
//	McAcpAxCycParID_2.VariableAddress := ADR(RPM);
//
//	MC_BR_CyclicProcessParID_AcpAx_3.Enable := TRUE;
//	MC_BR_CyclicProcessParID_AcpAx_3.Axis := ADR(Cutter);
//	MC_BR_CyclicProcessParID_AcpAx_3.DataAddress := ADR(McAcpAxCycParID_3);
//	MC_BR_CyclicProcessParID_AcpAx_3.Mode := mcACPAX_CYCLIC_PARID_READ;
//	MC_BR_CyclicProcessParID_AcpAx_3.NumberOfParIDs := 1;
//
//	McAcpAxCycParID_3.DataType:= mcACPAX_PARTYPE_REAL;
//	McAcpAxCycParID_3.ParID := 7760;//423 Actual Position, 246 Actual Position per Revolution
//	McAcpAxCycParID_3.RefreshMode := mcACPAX_CYCLIC_EVERY_RECORD;
//	McAcpAxCycParID_3.VariableAddress := ADR(ProductionSpeed);

//	MC_BR_CyclicProcessParID_AcpAx_2();
//	MC_BR_CyclicProcessParID_AcpAx_3();

END_ACTION
```

#### InitAxis.st
```iecst
ACTION InitAxis:

	MachineInitializing := TRUE;

	IF MpAxisBasic_Cutter.Info.ReadyToPowerOn THEN

		MpAxisBasic_Cutter.Power := TRUE;
		MachineInitializing := FALSE;

	END_IF;

	IF MpAxisBasic_Cutter.PowerOn AND NOT MpAxisBasic_Cutter.IsHomed THEN

		ReadyToInitHome := TRUE;
		ReadyToPower := FALSE;

	END_IF;

	IF ReadyToInitHome THEN

		MC_BR_InitHome_AcpAx_0.Execute := TRUE;

		IF MC_BR_InitHome_AcpAx_0.Done THEN
			MC_BR_InitHome_AcpAx_0.Execute := FALSE;
			ReadyToHome := TRUE;
			ReadyToInitHome := FALSE;
		END_IF;

		MC_BR_InitHome_AcpAx_0();

	END_IF;

	IF ReadyToHome AND (MpAxisBasic_Cutter.Info.PLCopenState = mcAXIS_STANDSTILL) THEN

		MachineHoming := TRUE;
		MpAxisBasic_Cutter.Home := TRUE;

		IF MpAxisBasic_Cutter.IsHomed THEN
			MachineHoming := FALSE;
			MpAxisBasic_Cutter.Home := FALSE;
			MODE_SELECTED := HMI_MODE_SELECTED;
			MachineReady := TRUE;
			ReadyToHome := FALSE;
		END_IF;

	END_IF;

	IF NOT (MpAxisBasic_Cutter.Info.DigitalInputsStatus.DriveEnable) THEN

		MpAxisBasic_Cutter.Stop := TRUE;
		MpAxisBasic_Cutter.Home := FALSE;
		MpAxisBasic_Cutter.AutoTune := FALSE;

	ELSE

		MpAxisBasic_Cutter.Stop := FALSE;

	END_IF;

END_ACTION
```

#### CountTurns.st
```iecst
ACTION CountTurns:

	CalculatedProductSpeed := (((HMICuttingLength/1000)*60)/MaxCount);

	IF (RealTurns ) >= (NeededTurns)  OR ManualCut OR EDGEPOS(oneCutEncoderCutterDieCmd) THEN
		ManualCut 		:= FALSE;
		auxToCut		:= FALSE;
		DelayTimer_0.IN := TRUE;
		MpAxisBasic_Cutter.MoveAdditive := TRUE;
		RelativeDistance	:=	((((HMICuttingLength/EncoderPerimeter)*Pulses)*CorrectionFactor) + ((CuttingOffset/EncoderPerimeter)*Pulses));
		NeededTurns := (RelativeDistance/Pulses) + RealTurns;
		CurrentProductTurns := 0;
		HMIRelativeDistanceOld := HMIRelativeDistance;
		HMIRelativeDistance	:=	((EncoderActPos) + ((HMICuttingLength/EncoderPerimeter)*Pulses));

	ELSE

		CurrentProductTurns := FullTurnCount + PartOfTurn;
	END_IF;

	EncoderActPosOld := EncoderActPos;

END_ACTION
```

### Data object Logical/AcpParTab (Apt)

#### AcpParTab.apt
```
AcoposParameterTable:
  Root Parameters:
    390 = 220 (Name=UDC_NOMINAL, Unit=V)  // CTRL DC bus: Nominal voltage
```

- Visualisation Logical/Visu_7inch (not shown)

- Visualisation Logical/VisuCtrl (not shown)

### Program Logical/ReadPar (IEC) - Este programa esta destinado para leer parametros del drive y desplegarlos a la visualización

#### ReadParameters.st - Implementation code
```iecst
(********************************************************************
 * COPYRIGHT -- Bernecker + Rainer
 ********************************************************************
 * Program: ReadParameters
 * File: ReadParameters.st
 * Author: murguiaj
 * Created: March 08, 2013
 ********************************************************************
 * Implementation of program ReadParameters
 ********************************************************************)

PROGRAM _INIT

(* TODO : Add your code here *)

END_PROGRAM

PROGRAM _CYCLIC

	MC_BR_CyclicProcessParID_AcpAx_0.Enable := EnablePar;
	MC_BR_CyclicProcessParID_AcpAx_0.Axis := ADR(Cutter);
	MC_BR_CyclicProcessParID_AcpAx_0.DataAddress := ADR(McAcpAxCycParID_0);
	MC_BR_CyclicProcessParID_AcpAx_0.Mode := ParIdAccessMode;//mcACPAX_CYCLIC_PARID_READ;
	MC_BR_CyclicProcessParID_AcpAx_0.NumberOfParIDs := 1;

	McAcpAxCycParID_0.DataType:= ParIdDataType;
	McAcpAxCycParID_0.ParID := motorTempParID; //381;
	McAcpAxCycParID_0.RefreshMode := mcACPAX_CYCLIC_EVERY_RECORD;
	McAcpAxCycParID_0.VariableAddress := ADR(motorTemp);

	MC_BR_CyclicProcessParID_AcpAx_1.Enable := TRUE;
	MC_BR_CyclicProcessParID_AcpAx_1.Axis := ADR(Cutter);
	MC_BR_CyclicProcessParID_AcpAx_1.DataAddress := ADR(McAcpAxCycParID_1);;
	MC_BR_CyclicProcessParID_AcpAx_1.NumberOfParIDs := 1;
	MC_BR_CyclicProcessParID_AcpAx_1.Mode := mcACPAX_CYCLIC_PARID_READ;

	McAcpAxCycParID_1.DataType:= ParIdDataType;
	McAcpAxCycParID_1.ParID := 377;
	McAcpAxCycParID_1.RefreshMode := mcACPAX_CYCLIC_EVERY_RECORD;
	McAcpAxCycParID_1.VariableAddress := ADR(cargaAcopos);

	MC_BR_CyclicProcessParID_AcpAx_0();
	MC_BR_CyclicProcessParID_AcpAx_1();

END_PROGRAM
```

#### ReadParameters.var - Local variables
```iecst
(********************************************************************
 * COPYRIGHT -- Bernecker + Rainer
 ********************************************************************
 * Program: ReadParameters
 * File: ReadParameters.var
 * Author: murguiaj
 * Created: March 08, 2013
 ********************************************************************
 * Local variables of program ReadParameters
 ********************************************************************)
VAR
	MC_BR_CyclicProcessParID_AcpAx_0 : MC_BR_CyclicProcessParID_AcpAx;
	MC_BR_CyclicProcessParID_AcpAx_1 : MC_BR_CyclicProcessParID_AcpAx;
	motorTemp : REAL;
	cargaAcopos : REAL;
	McAcpAxCycParID_0 : McAcpAxCycParIDType;
	McAcpAxCycParID_1 : McAcpAxCycParIDType;
	motorTempParID : UINT := 381;
	ParIdAccessMode : McAcpAxCycParIDModeEnum := mcACPAX_CYCLIC_PARID_READ;
	ParIdDataType : McAcpAxDataTypeEnum := mcACPAX_PARTYPE_REAL;
	EnablePar : BOOL := TRUE;
END_VAR
```

- Visualisation Logical/Visu (not shown)

### Program Logical/DataHandling/IMA_Client (IEC) - IMA client program

#### IMA_Client.st - IMA Client Implementation
```iecst
(********************************************************************
 * COPYRIGHT -- AutoMate MX
 ********************************************************************
 * Program: IMA_Client
 * File: IMA_Client.st
 * Author: Erick Alcantar
 * Created: July 8, 2024/9:54 PM
 ********************************************************************
 * Implementation of program IMA_Client
 ********************************************************************)

PROGRAM _INIT

	(*IMA Init*)
	pDatObjName := ADR('DataMap');
	statusInit := IMAinit(pDatObjName, errorInfo, ADR(stationId));
	(* Enabling connection automatically every boot-up *)
	enableConnection := TRUE;

END_PROGRAM

PROGRAM _CYCLIC

	CASE DataCollectorState OF

		ST_IDLE:
			(*IMA Communication*)
			IF (statusInit = IMA_OK) AND enableConnection THEN
				DataCollectorState := ST_CONNECTING;
			END_IF;

		ST_CONNECTING:
			statusComm := IMAcomm(stationId, connInfoPV, connInfoAUX);
			IF  connInfoPV.connectionStatus = IMA_OK THEN
				DataCollectorState := ST_CONNECTED;
			END_IF;

		ST_CONNECTED:
			statusComm := IMAcomm(stationId, connInfoPV, connInfoAUX);
			IF statusComm <> 0 THEN
				DataCollectorState := ST_ERROR_ACTIVE;
			ELSIF NOT enableConnection THEN
				DataCollectorState := ST_CLOSE_CONNECTION;
			END_IF

		ST_CLOSE_CONNECTION:
			statusClose := IMAclose(stationId);
			IF statusClose = 0 THEN
	  			DataCollectorState := ST_IDLE;
			END_IF;

		ST_ERROR_ACTIVE:

			timeOutConnection (IN := TRUE, PT := T#5s);

			IF resetError OR timeOutConnection.Q THEN
				statusClose 				:= IMAclose(stationId);
				IF statusClose = 0 THEN
					timeOutConnection.IN 	:= FALSE;
					DataCollectorState 		:= ST_RESET_ERROR;
				END_IF
			END_IF

		ST_RESET_ERROR:
			IF statusClose = 0 THEN
				resetError := FALSE;
				statusInit := IMAinit(pDatObjName, errorInfo, ADR(stationId));
				DataCollectorState := ST_IDLE;
			END_IF

	END_CASE;

	timeOutConnection();

END_PROGRAM

PROGRAM _EXIT

	//Close connection
	IMAclose(stationId);
	//Re-init
	pDatObjName := ADR('DataMap');
	statusInit := IMAinit(pDatObjName, errorInfo, ADR(stationId));

END_PROGRAM
```

#### IMA_Client.var - Local variables
```iecst
(********************************************************************
 * COPYRIGHT -- Bernecker + Rainer
 ********************************************************************
 * Program: IMA_Client
 * File: IMA_Client.var
 * Author: Bernecker + Rainer
 * Created: July 17, 2009
 ********************************************************************
 * Local variables of program IMA_Client
 ********************************************************************)
VAR
	pDatObjName : UDINT; (*Address of the name of the configuration data object*)
	statusInit : UINT; (*init status*)
	errorInfo : imaInfoStruct; (*Structure for outputting error information
*)
	stationId : UDINT; (*identifier used to reference and follow-up on a client/server communication instance
*)
	statusComm : UINT; (*communication status*)
	connInfoPV : imaInfoStruct; (*connection status and error information for variable services
*)
	connInfoAUX : imaInfoStruct; (*Structure for outputting connection status and error information for other services
*)
	statusClose : UINT; (*status of close *)
END_VAR
(******************************************* Data Collector variables *********************************************************)
VAR
	DataCollectorState : DataCollector_state_enum;
	enableConnection : BOOL;
	resetError : BOOL;
	timeOutConnection : TON;
END_VAR
```

### Program Logical/DataHandling/VarExchange (IEC) - Variable exchange progra,

#### variables.st - Implementation code
```iecst
(*********************************************************************************
 * Copyright: AutoMate MX
 * Author: Erick Alcantar
 * Created:   July 8, 2024/9:54 PM
 *********************************************************************************
  Programa para procesar las variables que son extraidas via INA2000 protocol
 *********************************************************************************)

PROGRAM _INIT

	(* Inicializando las variables declaradas en el DataMap*)
	actPosExtEncoder;
	cutEnabled;

END_PROGRAM

PROGRAM _CYCLIC

(* TODO : Add your code here *)

END_PROGRAM
```

### Data object Logical/DataHandling/DataMap (Simple) - configuration dataobject

#### DataMap.dat - AsIMA Configuration Data Object for STATION1
```
(********************************************************************
 * COPYRIGHT -- AutoMate MX
 ********************************************************************
 * Data object: DataMap
 * File: DataMap.dat
 * Author: Erick Alcantar
 * Created: July 17, 2009
 ********************************************************************
 * Data object para mapear las variables que se intercambiaran por
 * INA2000 protocol. Se declaran los paths hacia las variables del
 * servidor (PLC B&R externo).
 ********************************************************************)
;------------------------------------------------------------------------------------------------
;AsIMA Configuration Data Object
;------------------------------------------------------------------------------------------------
"[ROUTING_PATH]" ;Section name must be enclosed in brackets (name can be anything)
"/SECTION=INTERFACE" ;Defines the section type
"/CN=IF2.3" ;Routing path to the server (IF2 on CP0410 via Ethernet to Node Number 1 -> Server) Warning:
;Node numbers must be specified in HEXADECIMAL!
"[PV_LIST_IO]" ;Section name must be enclosed in brackets (name can be anything)
"/SECTION=PV" ;Defines the section type
"/SV=READ /SERVPV=ExternalEn:MpAxisBasic_externalEncoder.Position /CLNTPV=::actPosExtEncoder"
"/SV=READ /SERVPV=::dieCutterCtrl.status.enableCutterMachine /CLNTPV=::cutEnabled"
"/SV=READ /SERVPV=ExternalEn:encoderActPosPerRev /CLNTPV=::encActPosPerRev"
"/SV=READ /SERVPV=ExternalEn:cutEncoderMode /CLNTPV=::oneCutEncoderCutterDieCmd"
"[PV_LIST_INFO]" ;Section name must be enclosed in brackets (name can be anything)
"/SECTION=PV" ;Defines the section type
"/SV=WRITE /SERVPV=ExternalEn:productLenghtCutter /CLNTPV=MotionCtrl:HMICuttingLength"
```
